(* 
:Description: This function block is base for all other digital devices.
*)
FUNCTION_BLOCK ABSTRACT FB_DigitalDevice IMPLEMENTS I_DigitalDevice
VAR
	sName : STRING; (* Name of digital device instance *)
	sModuleType : STRING;
	sPortID		: STRING;
END_VAR
(*
Version history:

+-------------+------------+----------------+----------+------------------------------------------+
|Date         | Version    | created under  | Author   | Remark                                   |
+=============+============+================+==========+==========================================+
|2022-01      | 1.0.0.0    | V3.1.4024.22   | ADBO     | Function block created                   |
+-------------+------------+----------------+----------+------------------------------------------+

*)

PROPERTY ModuleType : REFERENCE TO STRING
GET
ModuleType REF= sModuleType;
END_GET
END_PROPERTY

METHOD MR_FirstCycle : BOOL
VAR_INPUT
	sName : STRING;
	sModuleType : STRING;
	sPortID		: STRING;
END_VAR
THIS^.sName := sName;
THIS^.sModuleType := sModuleType;
THIS^.sPortID := sPortID;
END_METHOD

PROPERTY Name : REFERENCE TO STRING
GET
Name REF= sName;
END_GET
END_PROPERTY

PROPERTY PortID : REFERENCE TO STRING
GET
PortID REF= sPortID;
END_GET
END_PROPERTY

END_FUNCTION_BLOCK

(* stored: Version 1.1.0.1, ProductVersion 3.1.4024.9
   POU FB_DigitalDevice: Id {91192233-2028-49cf-ab12-85fcaeefeda5}, SpecialFunc None
   Folder FirstCycle: Id {1c8c5f98-209a-402e-9e88-cc7599942cf8}
   Folder Properties: Id {e6f14551-760e-41fc-b0cf-38d01aae9c89}
   Property ModuleType: Id {6581fad5-7877-4e69-9424-376f13cdba42}
   Get Get: Id {f7811120-40e2-4b3a-bb81-b54e68f6afa0}
   Method MR_FirstCycle: Id {1cf68bcf-6260-4706-8c9b-4da8df45299d}
   Property Name: Id {4fbc2781-2f66-4ab0-9f22-21b3974ee3e2}
   Get Get: Id {af7b7a66-6c11-44b1-b409-95b6ec8f7e03}
   Property PortID: Id {af872da2-e47c-41ef-a147-62aeb27290ab}
   Get Get: Id {607b2655-6aef-4ce3-bf96-e041389e65b1} *)
